FUNCTION_BLOCK DIFF_EQUATION
  (* Standard: 61499-2 *)
  (* Version 2013_12_10, Gabriel *)
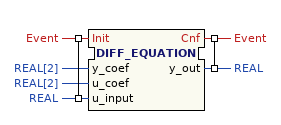
  EVENT_INPUT
    Init WITH u_input;
  END_EVENT
  EVENT_OUTPUT
    Cnf WITH y_out;
  END_EVENT
  VAR_INPUT
    y_coef : ARRAY [0..1] OF REAL;
    u_coef : ARRAY [0..1] OF REAL;
    u_input : REAL;
  END_VAR
  VAR_OUTPUT
    y_out : REAL;
  END_VAR
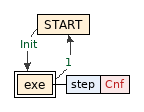
  EC_STATES
    exe : step -> Cnf;
    START;
  END_STATES
  EC_TRANSITIONS
    START TO exe := Init;
    exe TO START := 1;
  END_TRANSITIONS
  ALGORITHM step IN Lua:
if type(u_q ~= 'table') then
	u_q = {0, 0}
	y_out=0
end

u_q[2] = u_q[1]
u_q[1] = u_input

y_out = (-y_coef[2]*y_out + u_coef[2]*u_q[2] + u_coef[1]*u_q[1])/y_coef[1]
print(y_out)
  END_ALGORITHM
END_FUNCTION_BLOCK
